// TIA Portal V17 export
// export: Created 2023-11-29T12:25:14.5243927Z, ExportSetting WithDefaults, DisplayName Totally Integrated Automation Portal, DisplayVersion V17, DisplayName TIA Portal Openness, DisplayVersion V17, DisplayName TIA Portal Teamcenter Gateway, DisplayVersion V17, DisplayName TIA Portal Version Control Interface, DisplayVersion V17, DisplayName STEP 7 Professional, DisplayVersion V17, DisplayName STEP 7 Safety, DisplayVersion V17, DisplayName WinCC Advanced / Unified PC, DisplayVersion V17
VAR_GLOBAL   // PLC tag table "Variablentabelle_1"
   BO AT %I20.0 : Bool;
   B1 AT %I20.1 : Bool;
   B2 AT %I20.2 : Bool;
   B3 AT %I20.3 : Bool;
   B4 AT %I20.4 : Bool;
   Rücksetztaster_eins AT %I20.5 : Bool;
   Y1 AT %Q20.0 : Bool;
   Y2 AT %Q20.1 : Bool;
   Tag_4 AT %Q20.2 : Bool;
END_VAR
